// TIA Portal V20 export
FUNCTION_BLOCK "GetIdentRf"   // FB96, SCL
// stored: Access Published, MemoryReserve 100, SetENOAutomatically false
   VAR_OUTPUT
      selectedRFID : USInt := 1;
      selectedAntena : USInt;
      error : Word;
   END_VAR
   VAR_IN_OUT
      identRfAllUnits : Array[*] of "typeIdentRf";   // HMI: motorstarter values
      IdentRfInterfaceHmi : "typeIdentRfHmi";
   END_VAR
   VAR
      statSelectedRfReader : USInt := 1;   // HMI: Angewählte Interface Schnittstelle (1..16) / HMI: Selected unit
      statSelectedAntena : USInt := 1;
   END_VAR
   VAR CONSTANT
      "INVALID RFID" : Word := 16#7001;   // non existant rfid
      "INVALID ANTENA" : Word := 16#7002;   // non existant antena
      OK : Word := 16#7000;
   END_VAR
BEGIN
   REGION BLOCK INFO HEADER
       //===============================================================================
       // Siemens AG / (c)Copyright 2024
       //-------------------------------------------------------------------------------
       // Title:            LAF_GetMotorstarterSignals
       // Comment/Function: This block reads diagnostic information of a Motorstarter depending
       //                   on the unit and Control Module selected in the HMI by the user.
       // Library/Family:   Automation Framework / Motorstarter Diagnostic
       // Author:           Siemens Digital Industries
       // Tested with:      S7-1517TF V3.1
       // Engineering:      TIA Portal V19
       // Restrictions:     
       //                   Required UDTs: LAF_typeDriveDiagConfig, LAF_typeDriveDiagInterfaceHmi
       // Requirements:     S7-1500(T), MC_Version V8.0
       //-------------------------------------------------------------------------------
       // Change log table:
       // Version  | Date       | Expert in charge        | Changes applied
       //----------|------------|-------------------------|-----------------------------
       // 01.00.00 | 05.06.2024 | SIMATIC Systems Support | First released version
       //===============================================================================
   END_REGION BLOCK INFO HEADER

   REGION DESCRIPTION
   (/*This block reads diagnostic information (control inputs and outputs) of a Motorstarter. 
   At runtime, this block is enabled when the ET200SP Motorstarter screen is shown in the HMI. 
   Based on the selected motorstarter object in the HMI by the user. The shown information in the HMI depends on the
   Unit and Cotrol Module selected.*/)
   END_REGION DESCRIPTION

   REGION INPUTS
       //working with static values to keep the last selected value when opening for the first time the screen  

       #statSelectedRfReader := #IdentRfInterfaceHmi.selectedRfReader;
       #statSelectedAntena := #IdentRfInterfaceHmi.selectedAntena;

   END_REGION INPUTS

   REGION ASSIGNING TEMPORARY VALUES
       // Statement section REGION
       IF #statSelectedRfReader <= "NO_OF_RF_IDENT_DEVICES" THEN
           IF #statSelectedAntena <= "NO_OF_RF_ANTENNA_DEVICES" THEN
               #IdentRfInterfaceHmi.rfReader.deviceName := #identRfAllUnits[#statSelectedRfReader].IdentRfAntena[#statSelectedAntena].deviceName;
               #IdentRfInterfaceHmi.rfReader.deviceType := #identRfAllUnits[#statSelectedRfReader].IdentRfAntena[#statSelectedAntena].deviceType;
               #IdentRfInterfaceHmi.rfReader.deviceId := #identRfAllUnits[#statSelectedRfReader].IdentRfAntena[#statSelectedAntena].deviceId;
               #IdentRfInterfaceHmi.rfReader.tagType := #identRfAllUnits[#statSelectedRfReader].IdentRfAntena[#statSelectedAntena].tagType;
               #IdentRfInterfaceHmi.rfReader.cameraMode := #identRfAllUnits[#statSelectedRfReader].IdentRfAntena[#statSelectedAntena].cameraMode;
               #IdentRfInterfaceHmi.rfReader.resultState := #identRfAllUnits[#statSelectedRfReader].IdentRfAntena[#statSelectedAntena].resultState;
               #IdentRfInterfaceHmi.rfReader.progNo := #identRfAllUnits[#statSelectedRfReader].IdentRfAntena[#statSelectedAntena].progNo;
               #IdentRfInterfaceHmi.rfReader.progNumberWrite := #identRfAllUnits[#statSelectedRfReader].IdentRfAntena[#statSelectedAntena].progNumberWrite;
               #IdentRfInterfaceHmi.rfReader.enablePushbutton := #identRfAllUnits[#statSelectedRfReader].IdentRfAntena[#statSelectedAntena].enablePushbutton;
               #IdentRfInterfaceHmi.rfReader.status := #identRfAllUnits[#statSelectedRfReader].IdentRfAntena[#statSelectedAntena].status;
               #IdentRfInterfaceHmi.rfReader.alarmCategorie := #identRfAllUnits[#statSelectedRfReader].IdentRfAntena[#statSelectedAntena].alarmCategorie;
               #IdentRfInterfaceHmi.rfReader.alarmNo := #identRfAllUnits[#statSelectedRfReader].IdentRfAntena[#statSelectedAntena].alarmNo;
               #IdentRfInterfaceHmi.rfReader.alarmCode := #identRfAllUnits[#statSelectedRfReader].IdentRfAntena[#statSelectedAntena].alarmCode;
               #IdentRfInterfaceHmi.rfReader.resultColor := #identRfAllUnits[#statSelectedRfReader].IdentRfAntena[#statSelectedAntena].resultColor;
               #IdentRfInterfaceHmi.rfReader.statusColorCode := #identRfAllUnits[#statSelectedRfReader].IdentRfAntena[#statSelectedAntena].statusColorCode;
               #IdentRfInterfaceHmi.rfReader.datRead1 := #identRfAllUnits[#statSelectedRfReader].IdentRfAntena[#statSelectedAntena].datRead1;
               #IdentRfInterfaceHmi.rfReader.datRead2 := #identRfAllUnits[#statSelectedRfReader].IdentRfAntena[#statSelectedAntena].datRead2;
               #IdentRfInterfaceHmi.rfReader.datRead3 := #identRfAllUnits[#statSelectedRfReader].IdentRfAntena[#statSelectedAntena].datRead3;
               #IdentRfInterfaceHmi.rfReader.datRead4 := #identRfAllUnits[#statSelectedRfReader].IdentRfAntena[#statSelectedAntena].datRead4;

               #identRfAllUnits[#statSelectedRfReader].IdentRfAntena[#statSelectedAntena].pushbutton := #IdentRfInterfaceHmi.rfReader.pushbutton;
               #identRfAllUnits[#statSelectedRfReader].IdentRfAntena[#statSelectedAntena].datWrite1 := #IdentRfInterfaceHmi.rfReader.datWrite1;
               #identRfAllUnits[#statSelectedRfReader].IdentRfAntena[#statSelectedAntena].datWrite2 := #IdentRfInterfaceHmi.rfReader.datWrite2;
               #identRfAllUnits[#statSelectedRfReader].IdentRfAntena[#statSelectedAntena].datWrite3 := #IdentRfInterfaceHmi.rfReader.datWrite3;
               #identRfAllUnits[#statSelectedRfReader].IdentRfAntena[#statSelectedAntena].datWrite4 := #IdentRfInterfaceHmi.rfReader.datWrite4;

               #error := #OK;
           ELSE
               #error := #"INVALID ANTENA";
           END_IF;

       ELSE
           #error := #"INVALID RFID";
       END_IF;

   END_REGION


   REGION OUTPUTS
       // Statement section REGION
       #selectedAntena := #statSelectedAntena;
       #selectedRFID := #statSelectedRfReader;
   END_REGION
END_FUNCTION_BLOCK
